TYPE T_PLCTPL_CTRL :
STRUCT
	nCommand:	E_PLCTPL_COMMAND	:= E_PLCTPL_COMMAND.NONE; (* See E_PLCTPL_COMMAND *)
	bExecute:	BOOL;
	
END_STRUCT
END_TYPE

(* stored: Version 1.1.0.1, ProductVersion 3.1.4022.16
   DUT T_PLCTPL_CTRL: Id {17405076-e76e-47ad-8e66-f8b937714847} *)
